// TIA Portal project "PLC Template v3.2" (V15.1)

(* hardware
DEVICE "S71500/ET200MP station_1"  S7-1500 station
   slot 0: "Rail_0"  Rack  6ES7 590-1***0-0AA0
   slot 1: "PLC_1"  CPU 1512C-1 PN  6ES7 512-1CK01-0AB0  V2.6
      slot 3: "CPU display_1"  6ES7591-1AA00-0AA0
DEVICE "SCALANCE XC-200"  SCALANCE X-Station
   slot 0: "SCALANCE X rack"  Rail
   slot 0: "switch_1"  SCALANCE XC208  6GK5 208-0BA00-2AC2  V4.0
DEVICE "ET 200SP station_1"  ET 200SP-Station
   slot 0: "Rack_0"  Rack  6ES5 710-8MAx1
   slot 0: "io device_1"  IM 155-6 PN/2 HF  6ES7 155-6AU01-0CN0  V4.2
   slot 1: "DQ 8x24VDC/0.5A HF_1"  DQ 8x24VDC/0.5A HF  6ES7 132-6BF00-0CA0  V2.0
      slot 1: "DQ 8x24VDC/0.5A HF_1"  DQ 8x24VDC/0.5A HF
   slot 2: "DQ 8x24VDC/0.5A HF_2"  DQ 8x24VDC/0.5A HF  6ES7 132-6BF00-0CA0  V2.0
      slot 1: "DQ 8x24VDC/0.5A HF_2"  DQ 8x24VDC/0.5A HF
   slot 3: "DI 8x24VDC HF_1"  DI 8x24VDC HF  6ES7 131-6BF00-0CA0  V2.0
      slot 1: "DI 8x24VDC HF_1"  DI 8x24VDC HF
   slot 4: "DI 8x24VDC HF_2"  DI 8x24VDC HF  6ES7 131-6BF00-0CA0  V2.0
      slot 1: "DI 8x24VDC HF_2"  DI 8x24VDC HF
   slot 5: "AI 2xU/I 2-,4-wire HS_1"  AI 2xU/I 2-,4-wire HS  6ES7 134-6HB00-0DA1  V2.0
      slot 1: "AI 2xU/I 2-,4-wire HS_1"  AI 2xU/I 2-,4-wire HS
   slot 6: "AI 2xU/I 2-,4-wire HS_2"  AI 2xU/I 2-,4-wire HS  6ES7 134-6HB00-0DA1  V2.0
      slot 1: "AI 2xU/I 2-,4-wire HS_2"  AI 2xU/I 2-,4-wire HS
   slot 7: "AQ 2xU/I HS_1"  AQ 2xU/I HS  6ES7 135-6HB00-0DA1  V2.0
      slot 1: "AQ 2xU/I HS_1"  AQ 2xU/I HS
   slot 8: "CM 4xIO-Link_1"  CM 4xIO-Link  6ES7 137-6BD00-0BA0  V2.2
      slot 1: "CM 4xIO-Link_1"  6ES7 137-6BD00-0BA0
   slot 9: "Server module_1"  Server module  6ES7 193-6PA00-0AA0  V1.1
      slot 1: "Server module_1"  Server module
   slot 127: "BA 2xRJ45"  BA 2xRJ45  6ES7 193-6AR00-0AA0  V0.0
      slot 1: "Port_1"  X1 P1 R  6ES7 193-6AR00-0AA0  V0.0
      slot 2: "Port_2"  X1 P2 R  6ES7 193-6AR00-0AA0  V0.0
*)

// ===== PLC "PLC_1"  CPU 1512C-1 PN =====

ORGANIZATION_BLOCK "Main"   // OB1, LAD, ProgramCycle
TITLE = "Main Program Sweep (Cycle)"
{ S7_Optimized_Access := 'TRUE' }
VERSION : 0.1
   VAR_INPUT
      Initial_Call : Bool;   // Initial call of this OB
      Remanence : Bool;   // =True, if remanent data are available
   END_VAR
BEGIN
END_ORGANIZATION_BLOCK